// TIA Portal V20 export
FUNCTION "History" : Void   // FC93, LAD
// stored: SetENOAutomatically false
BEGIN

REGION Network 1: Call LER_visionHistory
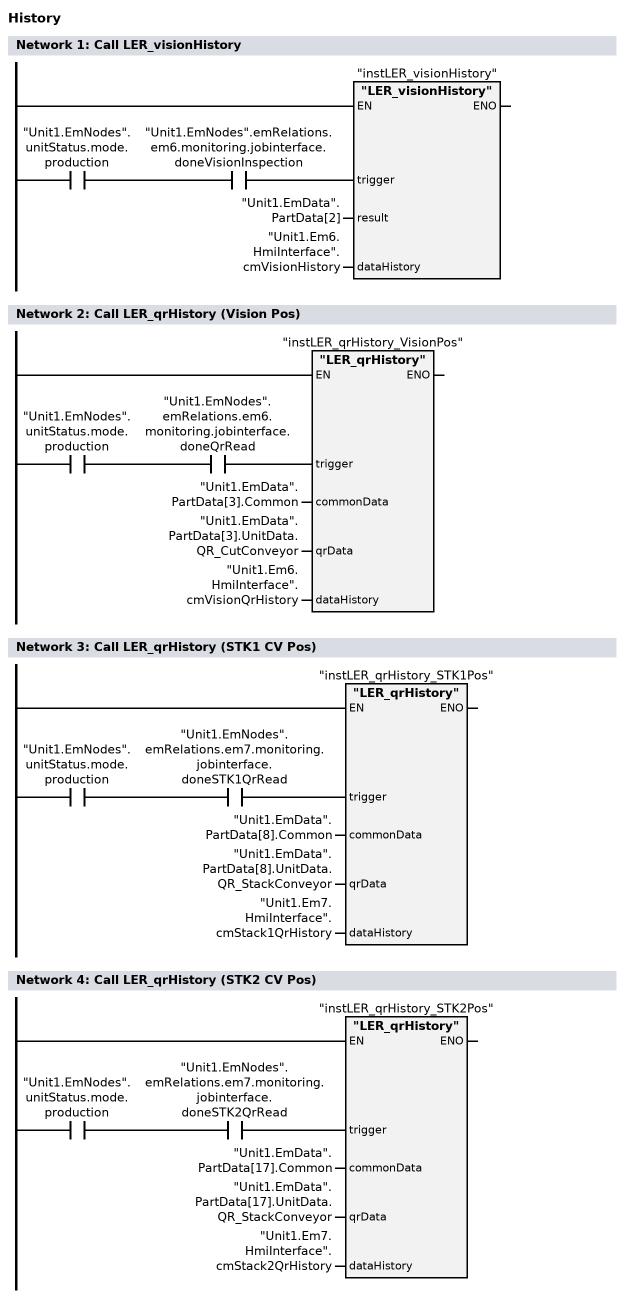
   RUNG wire#powerrail
      "instLER_visionHistory"(trigger := wire#w1, result := "Unit1.EmData".PartData[2], dataHistory := "Unit1.Em6.HmiInterface".cmVisionHistory)
   END_RUNG
   RUNG wire#powerrail
      Contact( "Unit1.EmNodes".unitStatus.mode.production )
      Contact( "Unit1.EmNodes".emRelations.em6.monitoring.jobinterface.doneVisionInspection )
   END_RUNG wire#w1
   // the same network as SCL:
   "instLER_visionHistory"(trigger := "Unit1.EmNodes".unitStatus.mode.production AND "Unit1.EmNodes".emRelations.em6.monitoring.jobinterface.doneVisionInspection,   // "LER_visionHistory"
                           result := "Unit1.EmData".PartData[2],
                           dataHistory := "Unit1.Em6.HmiInterface".cmVisionHistory);
END_REGION

REGION Network 2: Call LER_qrHistory (Vision Pos)
   RUNG wire#powerrail
      "instLER_qrHistory_VisionPos"(trigger := wire#w1, commonData := "Unit1.EmData".PartData[3].Common, qrData := "Unit1.EmData".PartData[3].UnitData.QR_CutConveyor, dataHistory := "Unit1.Em6.HmiInterface".cmVisionQrHistory)
   END_RUNG
   RUNG wire#powerrail
      Contact( "Unit1.EmNodes".unitStatus.mode.production )
      Contact( "Unit1.EmNodes".emRelations.em6.monitoring.jobinterface.doneQrRead )
   END_RUNG wire#w1
   // the same network as SCL:
   "instLER_qrHistory_VisionPos"(trigger := "Unit1.EmNodes".unitStatus.mode.production AND "Unit1.EmNodes".emRelations.em6.monitoring.jobinterface.doneQrRead,   // "LER_qrHistory"
                           commonData := "Unit1.EmData".PartData[3].Common,
                           qrData := "Unit1.EmData".PartData[3].UnitData.QR_CutConveyor,
                           dataHistory := "Unit1.Em6.HmiInterface".cmVisionQrHistory);
END_REGION

REGION Network 3: Call LER_qrHistory (STK1 CV Pos)
   RUNG wire#powerrail
      "instLER_qrHistory_STK1Pos"(trigger := wire#w1, commonData := "Unit1.EmData".PartData[8].Common, qrData := "Unit1.EmData".PartData[8].UnitData.QR_StackConveyor, dataHistory := "Unit1.Em7.HmiInterface".cmStack1QrHistory)
   END_RUNG
   RUNG wire#powerrail
      Contact( "Unit1.EmNodes".unitStatus.mode.production )
      Contact( "Unit1.EmNodes".emRelations.em7.monitoring.jobinterface.doneSTK1QrRead )
   END_RUNG wire#w1
   // the same network as SCL:
   "instLER_qrHistory_STK1Pos"(trigger := "Unit1.EmNodes".unitStatus.mode.production AND "Unit1.EmNodes".emRelations.em7.monitoring.jobinterface.doneSTK1QrRead,   // "LER_qrHistory"
                           commonData := "Unit1.EmData".PartData[8].Common,
                           qrData := "Unit1.EmData".PartData[8].UnitData.QR_StackConveyor,
                           dataHistory := "Unit1.Em7.HmiInterface".cmStack1QrHistory);
END_REGION

REGION Network 4: Call LER_qrHistory (STK2 CV Pos)
   RUNG wire#powerrail
      "instLER_qrHistory_STK2Pos"(trigger := wire#w1, commonData := "Unit1.EmData".PartData[17].Common, qrData := "Unit1.EmData".PartData[17].UnitData.QR_StackConveyor, dataHistory := "Unit1.Em7.HmiInterface".cmStack2QrHistory)
   END_RUNG
   RUNG wire#powerrail
      Contact( "Unit1.EmNodes".unitStatus.mode.production )
      Contact( "Unit1.EmNodes".emRelations.em7.monitoring.jobinterface.doneSTK2QrRead )
   END_RUNG wire#w1
   // the same network as SCL:
   "instLER_qrHistory_STK2Pos"(trigger := "Unit1.EmNodes".unitStatus.mode.production AND "Unit1.EmNodes".emRelations.em7.monitoring.jobinterface.doneSTK2QrRead,   // "LER_qrHistory"
                           commonData := "Unit1.EmData".PartData[17].Common,
                           qrData := "Unit1.EmData".PartData[17].UnitData.QR_StackConveyor,
                           dataHistory := "Unit1.Em7.HmiInterface".cmStack2QrHistory);
END_REGION
END_FUNCTION
